FUNCTION_BLOCK FB_Homing_StandardNC EXTENDS FB_Homing_Base IMPLEMENTS I_MotionSequence
VAR
    fbMcHome           : MC_Home;
    fbMoveAbs          : MC_MoveAbsolute;
    _ReferencePosition : LREAL;	
END_VAR
VAR_INPUT
bSensorInput :BOOL;	
END_VAR

METHOD Abort
VAR_INPUT
END_VAR
fbMcHome(Axis := _Axis.Axis, Execute := FALSE);
fbMoveAbs(Axis := _Axis.Axis, Execute := FALSE);
_bBusy := FALSE;
nStep := 0;
END_METHOD

METHOD CyclicLogic
CASE nStep OF
    0: 
        fbMcHome(Axis := _Axis.Axis, Execute := FALSE);
        fbMoveAbs(Axis := _Axis.Axis, Execute := FALSE);

    10: 
        fbMcHome(
            Axis            := _Axis.Axis, 
            Execute         := TRUE, 
            HomingMode      := MC_DefaultHoming,
            bCalibrationCam := bSensorInput
        );
        
        IF fbMcHome.Busy THEN
            nStep := 20;
        ELSIF fbMcHome.Error THEN
            nStep := 99;
        END_IF

    20: 
        fbMcHome(
            Axis            := _Axis.Axis,
            bCalibrationCam := bSensorInput 
        );
        
        IF fbMcHome.Done THEN
            fbMcHome(Axis := _Axis.Axis, Execute := FALSE);
            nStep := 30; 
        ELSIF fbMcHome.Error THEN
            nStep := 99;
        END_IF

    30: 
        fbMoveAbs(
            Axis     := _Axis.Axis,
            Execute  := TRUE,
            Position := _ReferencePosition,
            Velocity := 10.0
        );

        IF fbMoveAbs.Done THEN
            fbMoveAbs(Axis := _Axis.Axis, Execute := FALSE);
            _bBusy := FALSE;
            _bDone := TRUE;
            nStep  := 0; 
        ELSIF fbMoveAbs.Error THEN
            nStep := 99;
        END_IF

    99: 
        _bBusy    := FALSE;
        _bError   := TRUE;
        
        IF fbMoveAbs.Error THEN
            _bErrorID := fbMoveAbs.ErrorID;
        ELSE
            _bErrorID := fbMcHome.ErrorID;
        END_IF
        
        nStep     := 0;
END_CASE
END_METHOD

PROPERTY ReferencePosition : LREAL
GET
ReferencePosition := _ReferencePosition;
END_GET
SET
_ReferencePosition := ReferencePosition;
END_SET
END_PROPERTY

END_FUNCTION_BLOCK

(* stored: Version 1.1.0.1, ProductVersion 3.1.4024.15
   POU FB_Homing_StandardNC: Id {a68036c7-0906-4add-a8ec-d72fc1d336c0}, SpecialFunc None
   Method Abort: Id {771dc933-2c39-43b9-9ff8-76313dbd940b}
   Method CyclicLogic: Id {3ee0a176-f137-4cd7-8aa9-6d46284035d2}
   Property ReferencePosition: Id {a840ab22-ae29-47b2-96e3-1c1ed24b7c71}
   Get Get: Id {f7e4d8b4-387e-4059-b3ff-8c42b3ba92b7}
   Set Set: Id {b72435c2-93e7-43f7-9d00-ee210aa35269} *)
